FUNCTION_BLOCK ab5 (* Ab5example *)
  (* Standard: 61499-2 *)
  (* Version 1.0, 2023-05-29, steph *)
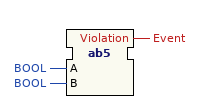
  EVENT_OUTPUT
    Violation;
  END_EVENT
  VAR_INPUT
    A : BOOL;
    B : BOOL;
  END_VAR
  VAR
    V : INT := 0;
  END_VAR
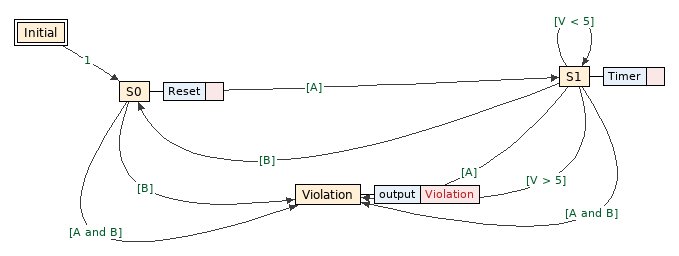
  EC_STATES
    Initial; (* Initial State *)
    S1 : Timer;
    Violation : output -> Violation;
    S0 : Reset;
  END_STATES
  EC_TRANSITIONS
    S1 TO Violation := [A];
    S1 TO S0 := [B];
    S0 TO S1 := [A];
    S0 TO Violation := [B];
    Initial TO S0 := 1;
    S1 TO Violation := [V > 5];
    S1 TO S1 := [V < 5];
    S0 TO Violation := [A and B];
    S1 TO Violation := [A and B];
  END_TRANSITIONS
  ALGORITHM Reset IN ST: (* Reset V to 0 *)
V := 0;
  END_ALGORITHM
  ALGORITHM Timer IN ST: (* counting V *)
V := V + 1;
  END_ALGORITHM
  ALGORITHM output IN ST: (* Violation *)

  END_ALGORITHM
END_FUNCTION_BLOCK
